// TIA Portal V20 export
// export: Created 2026-07-16T15:44:27.1761837Z, ExportSetting WithDefaults, DisplayName Totally Integrated Automation Portal, DisplayVersion V20 Update 5, DisplayName TIA Portal Openness, DisplayVersion V20 Update 4, DisplayName TIA Portal Version Control Interface, DisplayVersion V20 Update 5, DisplayName SINAMICS Startdrive Advanced, DisplayVersion V20, DisplayName SINAMICS DCC, DisplayVersion V20, DisplayName SINAMICS Startdrive G130, G150, S120, S150, SINAMICS MV, G220, S200, S210, DisplayVersion V20, DisplayName SINAMICS Startdrive G110M, G120, G120C, G120D, G120P, G115D, DisplayVersion V20, DisplayName STEP 7 Professional, DisplayVersion V20 Update 5, DisplayName STEP 7 Safety, DisplayVersion V20 Update 2, DisplayName WinCC Basic/Comfort/Advanced, DisplayVersion V20 Update 5, DisplayName WinCC Unified, DisplayVersion V20 Update 5
FUNCTION "FC_Inputs" : Void   // FC1, LAD
TITLE = Input Map
{ S7_Optimized_Access := 'TRUE' }
VERSION : 0.1
// stored: AutoNumber true, IsIECCheckEnabled false, SetENOAutomatically false, UDAEnableTagReadback false
BEGIN

REGION Network 1: PLC1 Built-in DI (CPU 1214C)
   // DI4_SYS_CycleStop is a normally-closed pushbutton: negated at this map layer so DB_Input.Cycle_Stop reads active-high (true = operator commanding stop) like every other buffer member - the input-mapping pattern's negated variant. Field polarity is absorbed here only; logic never compensates (C-304).
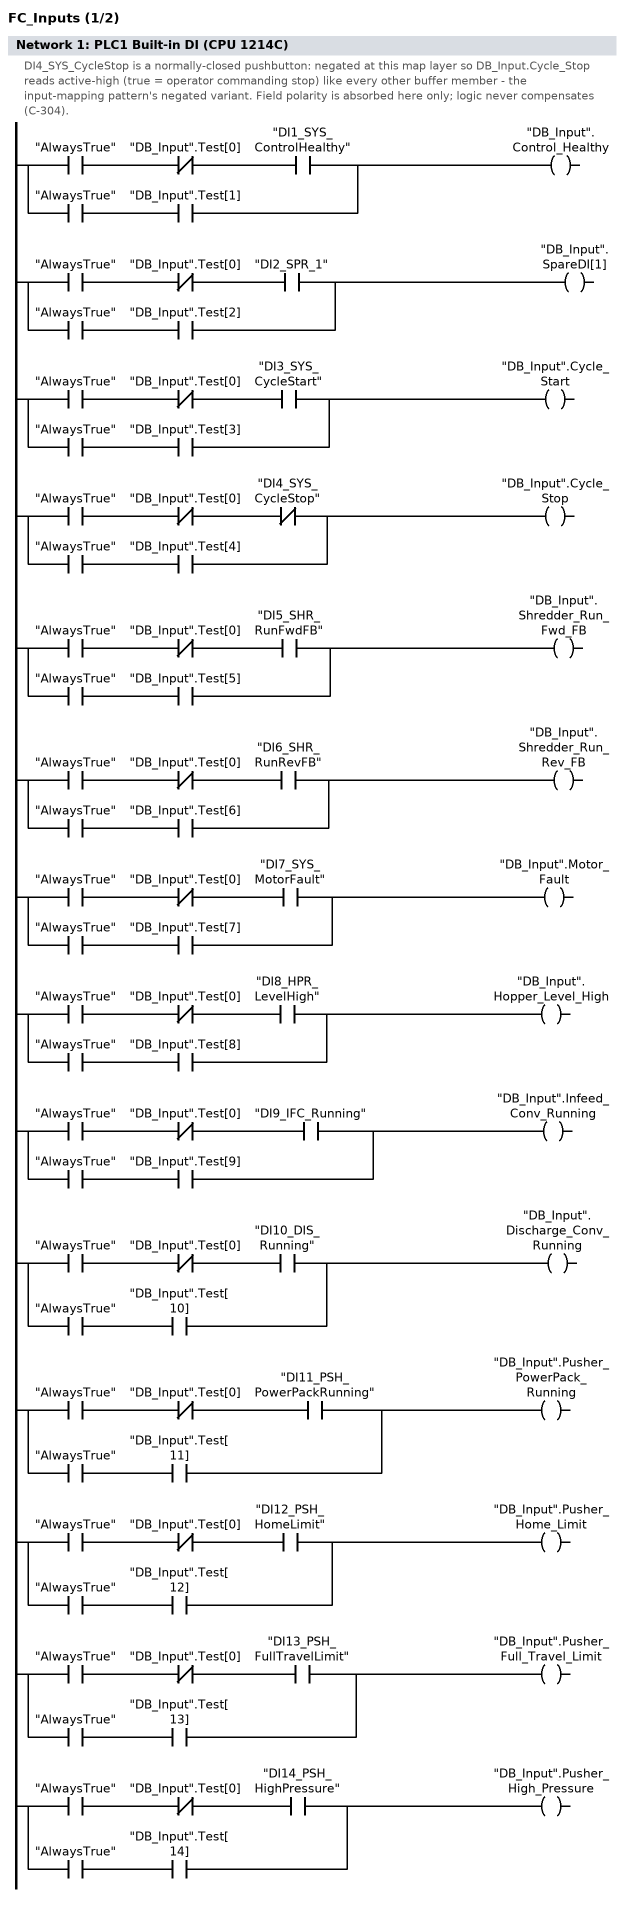
   RUNG wire#powerrail
      Contact( "AlwaysTrue" )
      I_Contact( "DB_Input".Test[0] )
      Contact( "DI1_SYS_ControlHealthy" )
      wire#w1
      Coil( "DB_Input".Control_Healthy )
   END_RUNG
   RUNG wire#powerrail
      Contact( "AlwaysTrue" )
      Contact( "DB_Input".Test[1] )
   END_RUNG wire#w1
   RUNG wire#powerrail
      Contact( "AlwaysTrue" )
      I_Contact( "DB_Input".Test[0] )
      Contact( "DI2_SPR_1" )
      wire#w2
      Coil( "DB_Input".SpareDI[1] )
   END_RUNG
   RUNG wire#powerrail
      Contact( "AlwaysTrue" )
      Contact( "DB_Input".Test[2] )
   END_RUNG wire#w2
   RUNG wire#powerrail
      Contact( "AlwaysTrue" )
      I_Contact( "DB_Input".Test[0] )
      Contact( "DI3_SYS_CycleStart" )
      wire#w3
      Coil( "DB_Input".Cycle_Start )
   END_RUNG
   RUNG wire#powerrail
      Contact( "AlwaysTrue" )
      Contact( "DB_Input".Test[3] )
   END_RUNG wire#w3
   RUNG wire#powerrail
      Contact( "AlwaysTrue" )
      I_Contact( "DB_Input".Test[0] )
      I_Contact( "DI4_SYS_CycleStop" )
      wire#w4
      Coil( "DB_Input".Cycle_Stop )
   END_RUNG
   RUNG wire#powerrail
      Contact( "AlwaysTrue" )
      Contact( "DB_Input".Test[4] )
   END_RUNG wire#w4
   RUNG wire#powerrail
      Contact( "AlwaysTrue" )
      I_Contact( "DB_Input".Test[0] )
      Contact( "DI5_SHR_RunFwdFB" )
      wire#w5
      Coil( "DB_Input".Shredder_Run_Fwd_FB )
   END_RUNG
   RUNG wire#powerrail
      Contact( "AlwaysTrue" )
      Contact( "DB_Input".Test[5] )
   END_RUNG wire#w5
   RUNG wire#powerrail
      Contact( "AlwaysTrue" )
      I_Contact( "DB_Input".Test[0] )
      Contact( "DI6_SHR_RunRevFB" )
      wire#w6
      Coil( "DB_Input".Shredder_Run_Rev_FB )
   END_RUNG
   RUNG wire#powerrail
      Contact( "AlwaysTrue" )
      Contact( "DB_Input".Test[6] )
   END_RUNG wire#w6
   RUNG wire#powerrail
      Contact( "AlwaysTrue" )
      I_Contact( "DB_Input".Test[0] )
      Contact( "DI7_SYS_MotorFault" )
      wire#w7
      Coil( "DB_Input".Motor_Fault )
   END_RUNG
   RUNG wire#powerrail
      Contact( "AlwaysTrue" )
      Contact( "DB_Input".Test[7] )
   END_RUNG wire#w7
   RUNG wire#powerrail
      Contact( "AlwaysTrue" )
      I_Contact( "DB_Input".Test[0] )
      Contact( "DI8_HPR_LevelHigh" )
      wire#w8
      Coil( "DB_Input".Hopper_Level_High )
   END_RUNG
   RUNG wire#powerrail
      Contact( "AlwaysTrue" )
      Contact( "DB_Input".Test[8] )
   END_RUNG wire#w8
   RUNG wire#powerrail
      Contact( "AlwaysTrue" )
      I_Contact( "DB_Input".Test[0] )
      Contact( "DI9_IFC_Running" )
      wire#w9
      Coil( "DB_Input".Infeed_Conv_Running )
   END_RUNG
   RUNG wire#powerrail
      Contact( "AlwaysTrue" )
      Contact( "DB_Input".Test[9] )
   END_RUNG wire#w9
   RUNG wire#powerrail
      Contact( "AlwaysTrue" )
      I_Contact( "DB_Input".Test[0] )
      Contact( "DI10_DIS_Running" )
      wire#w10
      Coil( "DB_Input".Discharge_Conv_Running )
   END_RUNG
   RUNG wire#powerrail
      Contact( "AlwaysTrue" )
      Contact( "DB_Input".Test[10] )
   END_RUNG wire#w10
   RUNG wire#powerrail
      Contact( "AlwaysTrue" )
      I_Contact( "DB_Input".Test[0] )
      Contact( "DI11_PSH_PowerPackRunning" )
      wire#w11
      Coil( "DB_Input".Pusher_PowerPack_Running )
   END_RUNG
   RUNG wire#powerrail
      Contact( "AlwaysTrue" )
      Contact( "DB_Input".Test[11] )
   END_RUNG wire#w11
   RUNG wire#powerrail
      Contact( "AlwaysTrue" )
      I_Contact( "DB_Input".Test[0] )
      Contact( "DI12_PSH_HomeLimit" )
      wire#w12
      Coil( "DB_Input".Pusher_Home_Limit )
   END_RUNG
   RUNG wire#powerrail
      Contact( "AlwaysTrue" )
      Contact( "DB_Input".Test[12] )
   END_RUNG wire#w12
   RUNG wire#powerrail
      Contact( "AlwaysTrue" )
      I_Contact( "DB_Input".Test[0] )
      Contact( "DI13_PSH_FullTravelLimit" )
      wire#w13
      Coil( "DB_Input".Pusher_Full_Travel_Limit )
   END_RUNG
   RUNG wire#powerrail
      Contact( "AlwaysTrue" )
      Contact( "DB_Input".Test[13] )
   END_RUNG wire#w13
   RUNG wire#powerrail
      Contact( "AlwaysTrue" )
      I_Contact( "DB_Input".Test[0] )
      Contact( "DI14_PSH_HighPressure" )
      wire#w14
      Coil( "DB_Input".Pusher_High_Pressure )
   END_RUNG
   RUNG wire#powerrail
      Contact( "AlwaysTrue" )
      Contact( "DB_Input".Test[14] )
   END_RUNG wire#w14
   // the same network as SCL:
   "DB_Input".Control_Healthy := ("AlwaysTrue" AND NOT "DB_Input".Test[0] AND "DI1_SYS_ControlHealthy") OR ("AlwaysTrue" AND "DB_Input".Test[1]);
   "DB_Input".SpareDI[1] := ("AlwaysTrue" AND NOT "DB_Input".Test[0] AND "DI2_SPR_1") OR ("AlwaysTrue" AND "DB_Input".Test[2]);
   "DB_Input".Cycle_Start := ("AlwaysTrue" AND NOT "DB_Input".Test[0] AND "DI3_SYS_CycleStart") OR ("AlwaysTrue" AND "DB_Input".Test[3]);
   "DB_Input".Cycle_Stop := ("AlwaysTrue" AND NOT "DB_Input".Test[0] AND NOT "DI4_SYS_CycleStop") OR ("AlwaysTrue" AND "DB_Input".Test[4]);
   "DB_Input".Shredder_Run_Fwd_FB := ("AlwaysTrue" AND NOT "DB_Input".Test[0] AND "DI5_SHR_RunFwdFB") OR ("AlwaysTrue" AND "DB_Input".Test[5]);
   "DB_Input".Shredder_Run_Rev_FB := ("AlwaysTrue" AND NOT "DB_Input".Test[0] AND "DI6_SHR_RunRevFB") OR ("AlwaysTrue" AND "DB_Input".Test[6]);
   "DB_Input".Motor_Fault := ("AlwaysTrue" AND NOT "DB_Input".Test[0] AND "DI7_SYS_MotorFault") OR ("AlwaysTrue" AND "DB_Input".Test[7]);
   "DB_Input".Hopper_Level_High := ("AlwaysTrue" AND NOT "DB_Input".Test[0] AND "DI8_HPR_LevelHigh") OR ("AlwaysTrue" AND "DB_Input".Test[8]);
   "DB_Input".Infeed_Conv_Running := ("AlwaysTrue" AND NOT "DB_Input".Test[0] AND "DI9_IFC_Running") OR ("AlwaysTrue" AND "DB_Input".Test[9]);
   "DB_Input".Discharge_Conv_Running := ("AlwaysTrue" AND NOT "DB_Input".Test[0] AND "DI10_DIS_Running") OR ("AlwaysTrue" AND "DB_Input".Test[10]);
   "DB_Input".Pusher_PowerPack_Running := ("AlwaysTrue" AND NOT "DB_Input".Test[0] AND "DI11_PSH_PowerPackRunning") OR ("AlwaysTrue" AND "DB_Input".Test[11]);
   "DB_Input".Pusher_Home_Limit := ("AlwaysTrue" AND NOT "DB_Input".Test[0] AND "DI12_PSH_HomeLimit") OR ("AlwaysTrue" AND "DB_Input".Test[12]);
   "DB_Input".Pusher_Full_Travel_Limit := ("AlwaysTrue" AND NOT "DB_Input".Test[0] AND "DI13_PSH_FullTravelLimit") OR ("AlwaysTrue" AND "DB_Input".Test[13]);
   "DB_Input".Pusher_High_Pressure := ("AlwaysTrue" AND NOT "DB_Input".Test[0] AND "DI14_PSH_HighPressure") OR ("AlwaysTrue" AND "DB_Input".Test[14]);
END_REGION

REGION Network 2: PLC1.1 SM1223 DI
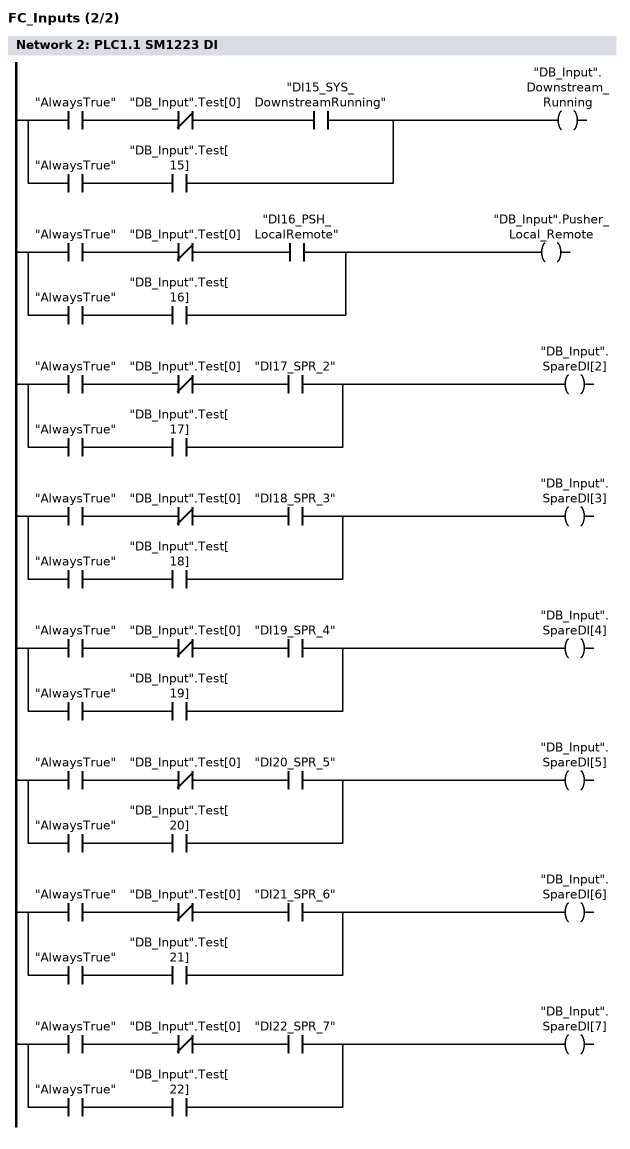
   RUNG wire#powerrail
      Contact( "AlwaysTrue" )
      I_Contact( "DB_Input".Test[0] )
      Contact( "DI15_SYS_DownstreamRunning" )
      wire#w1
      Coil( "DB_Input".Downstream_Running )
   END_RUNG
   RUNG wire#powerrail
      Contact( "AlwaysTrue" )
      Contact( "DB_Input".Test[15] )
   END_RUNG wire#w1
   RUNG wire#powerrail
      Contact( "AlwaysTrue" )
      I_Contact( "DB_Input".Test[0] )
      Contact( "DI16_PSH_LocalRemote" )
      wire#w2
      Coil( "DB_Input".Pusher_Local_Remote )
   END_RUNG
   RUNG wire#powerrail
      Contact( "AlwaysTrue" )
      Contact( "DB_Input".Test[16] )
   END_RUNG wire#w2
   RUNG wire#powerrail
      Contact( "AlwaysTrue" )
      I_Contact( "DB_Input".Test[0] )
      Contact( "DI17_SPR_2" )
      wire#w3
      Coil( "DB_Input".SpareDI[2] )
   END_RUNG
   RUNG wire#powerrail
      Contact( "AlwaysTrue" )
      Contact( "DB_Input".Test[17] )
   END_RUNG wire#w3
   RUNG wire#powerrail
      Contact( "AlwaysTrue" )
      I_Contact( "DB_Input".Test[0] )
      Contact( "DI18_SPR_3" )
      wire#w4
      Coil( "DB_Input".SpareDI[3] )
   END_RUNG
   RUNG wire#powerrail
      Contact( "AlwaysTrue" )
      Contact( "DB_Input".Test[18] )
   END_RUNG wire#w4
   RUNG wire#powerrail
      Contact( "AlwaysTrue" )
      I_Contact( "DB_Input".Test[0] )
      Contact( "DI19_SPR_4" )
      wire#w5
      Coil( "DB_Input".SpareDI[4] )
   END_RUNG
   RUNG wire#powerrail
      Contact( "AlwaysTrue" )
      Contact( "DB_Input".Test[19] )
   END_RUNG wire#w5
   RUNG wire#powerrail
      Contact( "AlwaysTrue" )
      I_Contact( "DB_Input".Test[0] )
      Contact( "DI20_SPR_5" )
      wire#w6
      Coil( "DB_Input".SpareDI[5] )
   END_RUNG
   RUNG wire#powerrail
      Contact( "AlwaysTrue" )
      Contact( "DB_Input".Test[20] )
   END_RUNG wire#w6
   RUNG wire#powerrail
      Contact( "AlwaysTrue" )
      I_Contact( "DB_Input".Test[0] )
      Contact( "DI21_SPR_6" )
      wire#w7
      Coil( "DB_Input".SpareDI[6] )
   END_RUNG
   RUNG wire#powerrail
      Contact( "AlwaysTrue" )
      Contact( "DB_Input".Test[21] )
   END_RUNG wire#w7
   RUNG wire#powerrail
      Contact( "AlwaysTrue" )
      I_Contact( "DB_Input".Test[0] )
      Contact( "DI22_SPR_7" )
      wire#w8
      Coil( "DB_Input".SpareDI[7] )
   END_RUNG
   RUNG wire#powerrail
      Contact( "AlwaysTrue" )
      Contact( "DB_Input".Test[22] )
   END_RUNG wire#w8
   // the same network as SCL:
   "DB_Input".Downstream_Running := ("AlwaysTrue" AND NOT "DB_Input".Test[0] AND "DI15_SYS_DownstreamRunning") OR ("AlwaysTrue" AND "DB_Input".Test[15]);
   "DB_Input".Pusher_Local_Remote := ("AlwaysTrue" AND NOT "DB_Input".Test[0] AND "DI16_PSH_LocalRemote") OR ("AlwaysTrue" AND "DB_Input".Test[16]);
   "DB_Input".SpareDI[2] := ("AlwaysTrue" AND NOT "DB_Input".Test[0] AND "DI17_SPR_2") OR ("AlwaysTrue" AND "DB_Input".Test[17]);
   "DB_Input".SpareDI[3] := ("AlwaysTrue" AND NOT "DB_Input".Test[0] AND "DI18_SPR_3") OR ("AlwaysTrue" AND "DB_Input".Test[18]);
   "DB_Input".SpareDI[4] := ("AlwaysTrue" AND NOT "DB_Input".Test[0] AND "DI19_SPR_4") OR ("AlwaysTrue" AND "DB_Input".Test[19]);
   "DB_Input".SpareDI[5] := ("AlwaysTrue" AND NOT "DB_Input".Test[0] AND "DI20_SPR_5") OR ("AlwaysTrue" AND "DB_Input".Test[20]);
   "DB_Input".SpareDI[6] := ("AlwaysTrue" AND NOT "DB_Input".Test[0] AND "DI21_SPR_6") OR ("AlwaysTrue" AND "DB_Input".Test[21]);
   "DB_Input".SpareDI[7] := ("AlwaysTrue" AND NOT "DB_Input".Test[0] AND "DI22_SPR_7") OR ("AlwaysTrue" AND "DB_Input".Test[22]);
END_REGION
END_FUNCTION
